TYPE STRING_5K : STRING(5000); END_TYPE

(* stored: Version 1.1.0.1, ProductVersion 3.1.4024.11
   DUT STRING_5K: Id {171bcfe8-4034-4fb2-8c68-3535e56f424b} *)
